Omron Sysmac Studio project CounterUP_DOWN (Sysmac Studio 1.65.0.64007, StandardProject)

# Controller new_Controller_0: NX1P2-1040DT1 version 1.69
Task PrimaryTask (priority 4, period or condition 2000): Program0



PROGRAM Program0
VAR
    deneme1 : BOOL;
    CTU1 : CTU;
    CTU_Reset : BOOL;
    CTU_PV : INT;
    CTU_CV : INT;
    deneme2 : BOOL;
    CTD1 : CTD;
    CTD_Load : BOOL;
    CTD_PV : INT;
    CTD_CV : INT;
    deneme3 : BOOL;
    CTUD1 : CTUD;
    CTUD_CD : BOOL;
    CTUD_Reset : BOOL;
    CTUD_Load : BOOL;
    CTUD_PV : INT;
    CTUD_QD : BOOL;
    CTUD_CV,CTD1 : INT;
    CTUD_CV : INT;
END_VAR
VAR
    _e1 : R_TRIG;
    _e2 : R_TRIG;
    _e3 : R_TRIG;
    _e4 : R_TRIG;
END_VAR

(* Section Section0: ladder, written here as Structured Text *)

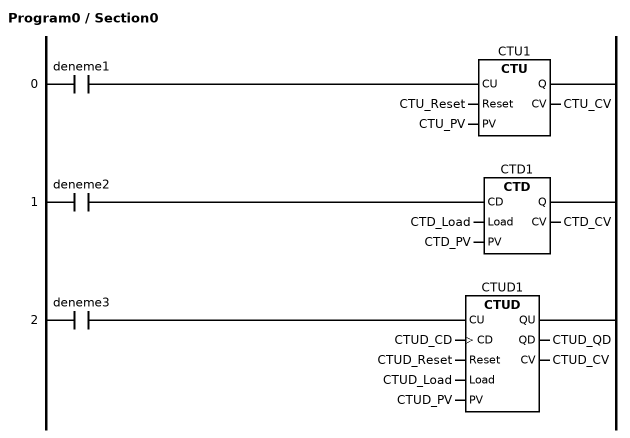
(* Rung 0 *)
_e1(CLK := deneme1);
CTU1(CU := _e1.Q, Reset := CTU_Reset, PV := CTU_PV, CV => CTU_CV);
(* Rung 1 *)
_e2(CLK := deneme2);
CTD1(CD := _e2.Q, Load := CTD_Load, PV := CTD_PV, CV => CTD_CV);
(* Rung 2 *)
_e3(CLK := CTUD_CD);
_e4(CLK := deneme3);
CTUD1(CU := _e4.Q, CD := _e3.Q, Reset := CTUD_Reset, Load := CTUD_Load, PV := CTUD_PV, QD => CTUD_QD, CV => CTUD_CV);
END_PROGRAM